Staubli VAL3: f1_cell_pick.pgx

program f1_cell_pick()
begin
  //pick from f1 put to bin
end
